FUNCTION_BLOCK FB_HSS
VAR_INPUT
END_VAR
VAR_OUTPUT
END_VAR
VAR
	//Properties
	bError 			: BOOL 				:= FALSE;
	eMode 			: E_ControlMode 	:= E_ControlMode.Off;	
	//Components
	//Valve
	fbValve 		:	FB_Valve_4_20A;
	//Pump with BACnet client
	fbPump 			:	FB_PumpBACnet2 :=(fbClient:=(nDeviceInstance:=16));
	//Temperature sensors
	fbTempSupPrim 	: 	FB_TempSensPt100;
	fbTempRetPrim 	: 	FB_TempSensPt100;
	fbTempSup 		: 	FB_TempSensPt100;
	fbTempRet 		: 	FB_TempSensPt100;
	//Controller
	fbControl 		: 	FB_HSSController;
	//Hydraulic circuit
	fbHydCir		: FB_HydMixCir := (	iPump 			:= fbPump,
										iValve			:= fbValve,
										iTempSupPrim 	:= fbTempSupPrim,
										iTempRetPrim 	:= fbTempRetPrim,
										iTempSup 		:= fbTempSup,
										iTempRet 		:= fbTempRet,
										iControl 		:= fbControl);
END_VAR

PROPERTY PUBLIC Error : BOOL
GET
Error := THIS^.bError;
END_GET
SET
THIS^.bError := Error;
END_SET
END_PROPERTY

PROPERTY PUBLIC Mode : E_ControlMode
GET
Mode := THIS^.eMode;
END_GET
SET
THIS^.eMode := Mode;
END_SET
END_PROPERTY

METHOD Run
VAR_INPUT
END_VAR
//Execute hydraulic circuit with its control routine
fbHydCir.Mode := eMode;
fbHydCir.Run();

//Write values to GVL
//Temperature datapoints
GVL.fHSSTempSupPrim 	:= fbTempSupPrim.Temperature;
GVL.fHSSTempRetPrim 	:= fbTempRetPrim.Temperature;
GVL.fHSSTempSup 		:= fbTempSup.Temperature;
GVL.fHSSTempRet 		:= fbTempRet.Temperature;
//ADS
ADS.fHSSTempSupPrimADS 	:= fbTempSupPrim.Temperature;
ADS.fHSSTempRetPrimADS 	:= fbTempRetPrim.Temperature;
ADS.fHSSTempSupADS 		:= fbTempSup.Temperature;
ADS.fHSSTempRetADS 		:= fbTempRet.Temperature;


//Valve datapoints
GVL.bHSSValveError 	:= fbValve.Error;
GVL.fHSSValveSet 		:= fbValve.OpeningSetpoint;
GVL.fHSSValveAct 		:= fbValve.OpeningActual;
//ADS
ADS.fHSSValveActADS 	:= fbValve.OpeningActual;


//Pump datapoints
GVL.eHSSPumpContMode	:= fbPump.ControlMode;
GVL.bHSSPumpError 		:= fbPump.Error;
GVL.bHSSPumpOperating	:= fbPump.Operating;
GVL.fHSSPumpPower		:= fbPump.PowerRating;
GVL.fHSSPumpPressure 	:= fbPump.Pressure;
GVL.bHSSPumpSetOn		:= fbPump.SetOn;
GVL.fHSSPumpSetpoint	:= fbPump.Setpoint;
GVL.fHSSPumpSpeed		:= fbPump.Speed;
GVL.fHSSPumpVolFlow	:= fbPump.VolumeFlow;
//ADS
ADS.bHSSPumpErrorADS 		:= fbPump.Error;
ADS.bHSSPumpOperatingADS	:= fbPump.Operating;
ADS.fHSSPumpPowerADS		:= fbPump.PowerRating;
ADS.fHSSPumpPressureADS 	:= fbPump.Pressure;
ADS.bHSSPumpSetOnADS		:= fbPump.SetOn;
ADS.fHSSPumpSpeedADS		:= fbPump.Speed;
ADS.fHSSPumpVolFlowADS		:= fbPump.VolumeFlow;
END_METHOD

PROPERTY PUBLIC TempRet : REAL
GET
TempRet:= THIS^.fbTempRet.TempRaw;
END_GET
SET
THIS^.fbTempRet.TempRaw := TempRet;
END_SET
END_PROPERTY

PROPERTY PUBLIC TempRetPrim : REAL
GET
TempRetPrim:= THIS^.fbTempRetPrim.TempRaw;
END_GET
SET
THIS^.fbTempRetPrim.TempRaw := TempRetPrim;
END_SET
END_PROPERTY

PROPERTY PUBLIC TempSup : REAL
GET
TempSup := THIS^.fbTempSup.TempRaw;
END_GET
SET
THIS^.fbTempSup.TempRaw := TempSup;
END_SET
END_PROPERTY

PROPERTY PUBLIC TempSupPrim : REAL
GET
TempSupPrim := THIS^.fbTempSupPrim.TempRaw;
END_GET
SET
THIS^.fbTempSupPrim.TempRaw := TempSupPrim;
END_SET
END_PROPERTY

PROPERTY PUBLIC Valve : REAL
GET
Valve := THIS^.fbValve.nOpeningAct;
END_GET
SET
THIS^.fbValve.nOpeningAct := Valve;
END_SET
END_PROPERTY

END_FUNCTION_BLOCK

(* stored: Version 1.1.0.1, ProductVersion 3.1.4024.3
   POU FB_HSS: Id {f613316f-4912-4f57-a234-55fa2c33a10a}, SpecialFunc None
   Property Error: Id {54c15d29-9597-417d-9336-3f1c72e395f4}
   Get Get: Id {33e45848-4417-41f9-a7c2-8ee070bc23bf}
   Set Set: Id {877eb2c9-1dc1-42f0-ad6e-6056f8e97d0a}
   Property Mode: Id {9ef373a3-05f4-40b5-9ff9-f7219466711f}
   Get Get: Id {5277489e-5a2c-4c6d-a112-29174d780764}
   Set Set: Id {29c0739e-0473-45be-8ffd-d53e17702b3c}
   Method Run: Id {0a45c8f2-945d-452f-aab3-9b4bc6b97b97}
   Property TempRet: Id {1b1a1b91-9d73-4bbc-8dec-ea9f717590b4}
   Get Get: Id {040325f7-b529-4c7c-805c-56e25c37ccae}
   Set Set: Id {c59cf482-93fb-4fa4-aa55-51b6ed2d345c}
   Property TempRetPrim: Id {36bad939-b4a4-4617-ad81-5856c9db414f}
   Get Get: Id {b6bd5173-6935-4781-889c-cee99e206eb8}
   Set Set: Id {33a96492-a8ad-48d5-b45c-9fffdfc1817e}
   Property TempSup: Id {e9cc9762-480d-4a6b-9f11-180c60a86692}
   Get Get: Id {8fa83531-82d0-43dc-9e4f-6a1b0b13a7b8}
   Set Set: Id {7214656d-cf9b-44af-a22c-6d1c181929ef}
   Property TempSupPrim: Id {99fdb839-1aea-4ece-98e8-28ccb92b41bc}
   Get Get: Id {4e2e9bc1-82c1-4ab8-8ec1-39f18b1133b2}
   Set Set: Id {481ccb78-11e9-46a4-a85d-9bfd5f14fd8f}
   Property Valve: Id {e4ec425f-4b0c-4d81-ae43-cb9479c3bc59}
   Get Get: Id {222b7711-c12d-45dc-a015-22c66df41b14}
   Set Set: Id {3d0f6c27-93d4-4c45-bc5b-b76d2dbcd8ec} *)
